(* CODESYS project bentonite_feeder

Project tree, tasks and I/O mapping:
  ecomatDisplay43inch_64bit_1 : ecomatDisplay43inch_64bit, ifm electronic, order no. 
      , version 3.5.19.4
    application Application
      libraries: CmpBitmapPool, * (System); ifmDevice_ecomatDisplay, * (ifm electronic); Datasource Symbolic Access, * (3S - Smart Software Solutions GmbH); Standard, 3.5.18.0 (System); Util, 3.5.19.0 (System)
      task control_task (cyclic, interval 2 ms, priority 17) calls control_prg
      task VISU_TASK (cyclic, interval 5 ms, priority 31) calls VisuElems.Visu_Prg, ifm_device
      control/
        function calc_smoothing [ST]
        program control_prg [CFC]
        function block fb_SlurryPump [LD]: calculate_time
        function block fb_TOI [ST]
        function block PV7603 [ST]
      hmi/
        d pad/
          function block d_pad_fb [ST]: down, left, right, switch_visu, up
        program ifm_device [ST]
        image pool ImagePool
        interfaces/
          function block selectable_item_base [ST]: hover, item_action, leave, select
        menu objects/
          dummy item/
            visualisation dummy_item
            function block fb_dummy_item [ST]: fb_Init, item_action
          hamburger/
            function block fb_hamburger_item [ST]: close, fb_Init, item_action
            visualisation hamburger
          menu data/
            visualisation Empty_visu_reference
            global variables g_menu_colors
            image pool menu_pool
            data type nav_item_enum
          menu item/
            function block fb_menu_item [ST]: fb_Init, item_action
            visualisation menu_item
          toggle items/
            integer setting/
              function block fb_integer_setting [ST]: decrease, fb_Init, increase, item_action, leave
              visualisation integer_setting_dialog
              visualisation integer_setting_item
            number selector/
            real setting/
              function block fb_real_setting [ST]: decrease, fb_Init, increase, item_action, leave
              visualisation real_setting_item
            visualisation toggle_item
        visualisation Parameters
        visualisation Test_Frame_2
        visualisation Test_Frame_3
        visualisation Test_Frame_4
        visualisation Test_Frame_5
        visualisation Test_Frame
      global variables pr
      visualisation Test_Visu
    Communication : Communication, ifm electronic, version 3.5.19.4
      CAN : CAN, ifm electronic, version 3.5.19.4
      Ethernet : Ethernet, ifm electronic, version 3.5.19.4
  5ce3da45-db07-42e7-a21c-a00fff4ed8f6|C:\Users\johnm\Downloads\Full-Circle-Logo-HorizStack.png
  5ce3da45-db07-42e7-a21c-a00fff4ed8f6|C:\Users\johnm\Downloads\Full-Circle-Logo-HorizStack.png
  5ce3da45-db07-42e7-a21c-a00fff4ed8f6|C:\Users\johnm\Full Circle Water\Controls - Documents\Software Versions\graphics\Full Circle Logos (new)\Horizontal\Full-Circle-Logo-Horizontal.png
  5ce3da45-db07-42e7-a21c-a00fff4ed8f6|C:\Users\johnm\Pictures\analytics icon.png
  5ce3da45-db07-42e7-a21c-a00fff4ed8f6|C:\Users\johnm\Pictures\analytics icon.png
  5ce3da45-db07-42e7-a21c-a00fff4ed8f6|C:\Users\johnm\Pictures\analytics icon.png
  5ce3da45-db07-42e7-a21c-a00fff4ed8f6|C:\Users\johnm\Pictures\analytics icon.png
  5ce3da45-db07-42e7-a21c-a00fff4ed8f6|C:\Users\johnm\Pictures\analytics icon.png
  5ce3da45-db07-42e7-a21c-a00fff4ed8f6|C:\Users\johnm\Pictures\analytics icon.png
  5ce3da45-db07-42e7-a21c-a00fff4ed8f6|C:\Users\johnm\Pictures\analytics icon.png
  text list GlobalTextList
  visualisation Visualization
*)

// ecomatDisplay43inch_64bit_1/Application/hmi/menu objects/menu data/nav_item_enum
{attribute 'qualified_only'}
{attribute 'strict'}
TYPE nav_item_enum :
(
	hover:= 0,
	select:= 1,
	selected:= 2,
	leave:= 3, 
	accent:= 4,
	alarm:= 5
);
END_TYPE

// ecomatDisplay43inch_64bit_1/Application/pr
{attribute 'qualified_only'}
VAR_GLOBAL PERSISTENT RETAIN
	//parameter list
	pump_gpm: UINT;
	dose_trigger: UINT; //gallons
	dose_amount: REAL; //pounds with 1 decimal
	charge_time: UINT; //time
	sensor_setpoint: UINT;
	psi_threshold: UINT;
	psi_debounce: UINT; //time
	flow_back: UINT; //amount of gal backfeeding on pump-off
END_VAR

// ecomatDisplay43inch_64bit_1/Application/hmi/menu objects/menu data/g_menu_colors
{attribute 'qualified_only'}
VAR_GLOBAL
	default: DWORD:= 16#FF2C323F;
	nav: ARRAY [nav_item_enum.hover..nav_item_enum.alarm] OF DWORD:= 
		[16#FF464C57, 16#FF7B7F87, 16#FF7B7F87, 16#FF2C323F, 16#FF89A1D3];
	//each position contains corresponding color
	//declare local variable of type 'nav_item_enum,' (ex. 'nav_command') and pass g_menu_colors.nav[nav_command] to the element
END_VAR

// ecomatDisplay43inch_64bit_1/Application/control/control_prg
PROGRAM control_prg
VAR
	simu_toi: fb_TOI; 
	simu_in: BOOL; 
	simu_reset: BOOL;
	tmr: TON; 
END_VAR

simu_toi(IN := simu_in, RESET := simu_reset, PT := T#20s); // FB_TOI

END_PROGRAM

// ecomatDisplay43inch_64bit_1/Application/control/fb_TOI
FUNCTION_BLOCK fb_TOI

VAR_INPUT
	IN: BOOL;
	RESET: BOOL;
	PT: TIME;
END_VAR

VAR_OUTPUT
	ET: TIME;
	Q: BOOL;
END_VAR

VAR
	Start_Time: TIME;
	Saved_Time: TIME;
	RT_IN: R_TRIG;
END_VAR

RT_IN(
	CLK:= IN,
	Q=>,
);

IF RESET THEN 
	ET:= T#0MS;
	Saved_Time:= T#0MS; //reset the time output
END_IF

IF RT_IN.Q THEN
	Start_Time:= TIME(); //when in triggers keep track of time
	Saved_Time:= ET; //and "save" the output time
END_IF

IF IN THEN
	ET:= Saved_Time + TIME() - Start_Time; 
END_IF //output time is saved time and counts from when IN triggered

Q:= ET >= PT; //q is true when output time is above PT

END_FUNCTION_BLOCK

// ecomatDisplay43inch_64bit_1/Application/hmi/ifm_device
PROGRAM ifm_device

VAR
	Reset_Keys: ifmDevice.ResetKeyMapping;
	Key_Map: ifmDevice.SetKeyMapping;
	KeyMapping: ifmDevice.stKEY_MAP_LIST;
	test: BOOL;
END_VAR

VAR
	Start_up_done: BOOL:= 0;
END_VAR

KeyMapping.eKey2_Up:=  		ifmDevice.eKEY_MAP_CODES.LEFT;
KeyMapping.eKey2_Down:=		ifmDevice.eKEY_MAP_CODES.RIGHT;
KeyMapping.eKey2_Left:=		ifmDevice.eKEY_MAP_CODES.DOWN;
KeyMapping.eKey2_Right:=	ifmDevice.eKEY_MAP_CODES.UP;
KeyMapping.eKey2_Return:=	ifmDevice.eKEY_MAP_CODES.SPACE;
		
Reset_Keys(
	xExecute:= NOT(Start_up_done AND test),
	xDone=>,
	xError=>,
	eDiagInfo=>
);

Key_Map(
	xExecute:= NOT(start_up_done AND test),
	xDone=>,
	xError=>,
	eDiagInfo=>,
	stKeyMapList:= KeyMapping,
);

test:= Start_up_done;
Start_up_done S= Reset_Keys.xDone AND Key_Map.xDone;

END_PROGRAM

// ecomatDisplay43inch_64bit_1/Application/control/calc_smoothing
FUNCTION calc_smoothing : REAL
VAR_INPUT
	cycle_time: TIME;
	time_constant: TIME:= T#2MS; 
END_VAR
VAR CONSTANT
	
END_VAR

calc_smoothing:= 1 - EXPT(2.71828, (-1.0 * (TO_REAL(cycle_time)) / TO_REAL(time_constant)));

END_FUNCTION

// ecomatDisplay43inch_64bit_1/Application/control/fb_SlurryPump
FUNCTION_BLOCK fb_SlurryPump

VAR_INPUT
	pumping: BOOL;
	gpm: UINT;
	trigger_volume: UINT;
END_VAR

VAR_OUTPUT
	dose: BOOL; //single shot
END_VAR

VAR
	flow_counter: REAL;
	time_val: TIME;
	timer_fb: fb_TOI;
END_VAR

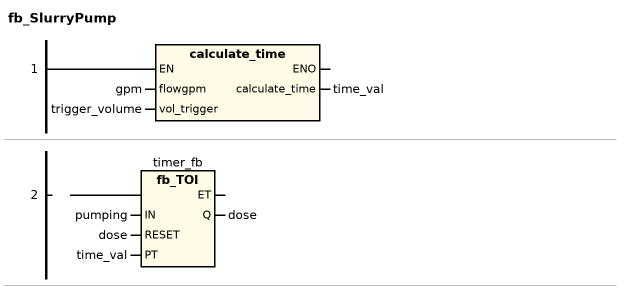
// NETWORK 1
time_val := calculate_time(flowgpm := gpm, vol_trigger := trigger_volume);

// NETWORK 2
timer_fb(IN := pumping, RESET := dose, PT := time_val, Q => dose); // fb_TOI

METHOD calculate_time : TIME
VAR_INPUT
	flowgpm: UINT;
	vol_trigger: UINT;
END_VAR

VAR CONSTANT
	min_to_ms: UINT:= 60000;
END_VAR
calculate_time:= TO_TIME(
	TO_UINT(
		TO_REAL(vol_trigger) 
	/ 	TO_REAL(flowgpm) //calc how many minutes
	* 	min_to_ms) //convert to ms
);
END_METHOD

END_FUNCTION_BLOCK

// ecomatDisplay43inch_64bit_1/Application/control/PV7603
FUNCTION_BLOCK PV7603
VAR_INPUT
	IOL_Read: ARRAY [0..3] OF WORD;
	time_setting: TIME;
END_VAR
VAR_OUTPUT
END_VAR
VAR
	factor: REAL;
	cycle_time: TIME;
	filtered_val: REAL;
	raw_signal: REAL;
END_VAR

raw_signal:= TO_REAL(IOL_Read[0]);

factor := calc_smoothing(T#2MS, time_setting);

filtered_val:= 
	(filtered_val * (1.0 - factor)) 
+ 	(raw_signal * factor);

END_FUNCTION_BLOCK

// ecomatDisplay43inch_64bit_1/Application/hmi/d pad/d_pad_fb
FUNCTION_BLOCK d_pad_fb
VAR_INPUT CONSTANT
	x_bounds: UINT:= 3;
END_VAR
VAR_INPUT
	disable_nav: BOOL;
	y_bounds: ARRAY [0..20] OF UINT;
END_VAR

VAR_OUTPUT
	position: ARRAY [0..1] OF UINT:= [1, 0];
END_VAR

METHOD down
VAR_INPUT
END_VAR
IF THIS^.disable_nav THEN
	RETURN; 
END_IF

IF THIS^.y_bounds[position[0]] > THIS^.position[1] THEN
	THIS^.position[1]:= THIS^.position[1] + 1;
END_IF
END_METHOD

METHOD left
VAR_INPUT
END_VAR
IF THIS^.disable_nav THEN
	RETURN; 
END_IF

IF THIS^.x_bounds > THIS^.position[0] THEN
	THIS^.position[0]:= THIS^.position[0] + 1;
	THIS^.position[1]:= 0;
END_IF
END_METHOD

METHOD right
VAR_INPUT
END_VAR
IF THIS^.disable_nav THEN
	RETURN; 
END_IF

IF THIS^.position[0] < 1 THEN
	RETURN;
END_IF

THIS^.position[0]:= THIS^.position[0] - 1;
THIS^.position[1]:= 0;
END_METHOD

METHOD switch_visu
VAR_INPUT
END_VAR
THIS^.position[0]:= 0;
THIS^.position[1]:= 0;
END_METHOD

METHOD up
VAR_INPUT
END_VAR
IF THIS^.disable_nav THEN
	RETURN; 
END_IF

IF THIS^.position[1] < 1 THEN
	RETURN;
END_IF

THIS^.position[1]:= THIS^.position[1] - 1;
END_METHOD

END_FUNCTION_BLOCK

// ecomatDisplay43inch_64bit_1/Application/hmi/interfaces/selectable_item_base
FUNCTION_BLOCK ABSTRACT selectable_item_base
VAR_INPUT
	position: ARRAY [0..1] OF UINT;
END_VAR
VAR_OUTPUT
END_VAR
VAR
	color: DWORD:= 16#FFFFFFFF;
END_VAR

METHOD hover
THIS^.color:= g_menu_colors.nav[nav_item_enum.hover];
//changes fb 'color' to menu color value for hover action
END_METHOD

METHOD ABSTRACT item_action
END_METHOD

METHOD leave
VAR_INPUT
END_VAR
THIS^.color:= g_menu_colors.nav[nav_item_enum.leave];
//changes fb 'color' to menu color value for hover action
END_METHOD

METHOD select
THIS^.color:= g_menu_colors.nav[nav_item_enum.select];
//changes fb 'color' to menu color value for selected action
THIS^.item_action();
END_METHOD

END_FUNCTION_BLOCK

// ecomatDisplay43inch_64bit_1/Application/hmi/menu objects/dummy item/fb_dummy_item
FUNCTION_BLOCK fb_dummy_item EXTENDS selectable_item_base
VAR_INPUT
END_VAR
VAR_OUTPUT
END_VAR
VAR
END_VAR

//FB_Init is always available implicitly and it is used primarily for initialization.
//The return value is not evaluated. For a specific influence, you can also declare the
//methods explicitly and provide additional code there with the standard initialization
//code. You can evaluate the return value.
METHOD FB_Init: BOOL
VAR_INPUT
    bInitRetains: BOOL; // TRUE: the retain variables are initialized (reset warm / reset cold)
    bInCopyCode: BOOL:= TRUE;  // TRUE: the instance will be copied to the copy code afterward (online change)   
END_VAR
THIS^.color:= g_menu_colors.default;
END_METHOD

METHOD item_action
END_METHOD

END_FUNCTION_BLOCK

// ecomatDisplay43inch_64bit_1/Application/hmi/menu objects/hamburger/fb_hamburger_item
FUNCTION_BLOCK fb_hamburger_item EXTENDS selectable_item_base
VAR_INPUT
END_VAR
VAR_OUTPUT
	open: BOOL;
END_VAR

METHOD close : BOOL
VAR_INPUT
END_VAR
THIS^.open:= 0;
END_METHOD

//FB_Init is always available implicitly and it is used primarily for initialization.
//The return value is not evaluated. For a specific influence, you can also declare the
//methods explicitly and provide additional code there with the standard initialization
//code. You can evaluate the return value.
METHOD FB_Init: BOOL
VAR_INPUT
    bInitRetains: BOOL; // TRUE: the retain variables are initialized (reset warm / reset cold)
    bInCopyCode: BOOL:= TRUE;  // TRUE: the instance will be copied to the copy code afterward (online change)   
END_VAR
THIS^.color:= g_menu_colors.default;
END_METHOD

METHOD item_action
THIS^.open:= 1;
END_METHOD

END_FUNCTION_BLOCK

// ecomatDisplay43inch_64bit_1/Application/hmi/menu objects/menu item/fb_menu_item
FUNCTION_BLOCK fb_menu_item	EXTENDS selectable_item_base
(*Visualizations of 'menu items,' code implementation using references contained here.*)
(*All implementation is done using the fb methods, and are called in visualization.*)
VAR_INPUT
	visu_reference: REFERENCE TO UINT;
	(*index of configured frame visu*)
	(*and order in list - d pad navigation*)
END_VAR
VAR_OUTPUT
END_VAR

//FB_Init is always available implicitly and it is used primarily for initialization.
//The return value is not evaluated. For a specific influence, you can also declare the
//methods explicitly and provide additional code there with the standard initialization
//code. You can evaluate the return value.
METHOD FB_Init: BOOL
VAR_INPUT
    bInitRetains: BOOL; // TRUE: the retain variables are initialized (reset warm / reset cold)
    bInCopyCode: BOOL:= TRUE;  // TRUE: the instance will be copied to the copy code afterward (online change)   
END_VAR
THIS^.color:= g_menu_colors.default;
END_METHOD

METHOD item_action
THIS^.visu_reference:= THIS^.position[1] - 1;
(*assign index to the frame*)
END_METHOD

END_FUNCTION_BLOCK

// ecomatDisplay43inch_64bit_1/Application/hmi/menu objects/toggle items/integer setting/fb_integer_setting
FUNCTION_BLOCK fb_integer_setting EXTENDS selectable_item_base
VAR_INPUT
	integer: REFERENCE TO UINT;
	increment: UINT;
	default: UINT;
	max_value: UINT;
	min_value: UINT;
END_VAR
VAR_OUTPUT
	selected: BOOL;

END_VAR
VAR
	int_array: ARRAY [0..4] OF UINT; // ones, tens, hundreds, thousands, ten-thousands
END_VAR

METHOD decrease
VAR_INPUT
END_VAR
IF THIS^.integer - THIS^.increment >= THIS^.min_value THEN
	THIS^.integer:= THIS^.integer - THIS^.increment;
END_IF
END_METHOD

(*FB_Init is always available implicitly and it is used primarily for initialization.
The return value is not evaluated. For a specific influence, you can also declare the
methods explicitly and provide additional code there with the standard initialization
code. You can evaluate the return value.*)
METHOD FB_Init : BOOL
VAR_INPUT
	(* TRUE: the retain variables are initialized (reset warm / reset cold)*)
	bInitRetains	: BOOL;
	(* TRUE: the instance will be copied to the copy code afterward (online change)   *)
	bInCopyCode	: BOOL := TRUE;
END_VAR
THIS^.color:= g_menu_colors.default;
(*
THIS^.int_array[0]:= THIS^.integer / 1		MOD 10;
THIS^.int_array[1]:= THIS^.integer / 10		MOD 10;
THIS^.int_array[2]:= THIS^.integer / 100	MOD 10;
THIS^.int_array[3]:= THIS^.integer / 1000	MOD 10;
THIS^.int_array[4]:= THIS^.integer / 10000	MOD 10;*)
END_METHOD

METHOD increase
VAR_INPUT
END_VAR
IF THIS^.integer + THIS^.increment <= THIS^.max_value THEN
	THIS^.integer:= THIS^.integer + THIS^.increment;
END_IF
END_METHOD

METHOD item_action
VAR_INPUT
END_VAR
THIS^.selected:= THIS^.selected XOR TRUE;
IF NOT THIS^.selected THEN
	THIS^.hover();
END_IF
END_METHOD

METHOD leave
VAR_INPUT
END_VAR
THIS^.color:= g_menu_colors.nav[nav_item_enum.leave];
//changes fb 'color' to menu color value for hover action
THIS^.selected:= 0;
END_METHOD

END_FUNCTION_BLOCK

// ecomatDisplay43inch_64bit_1/Application/hmi/menu objects/toggle items/real setting/fb_real_setting
FUNCTION_BLOCK fb_real_setting EXTENDS selectable_item_base
VAR_INPUT
	real_var: REFERENCE TO REAL;
	increment: REAL;
	max_value: REAL;
	min_value: REAL;
END_VAR
VAR_OUTPUT
	selected: BOOL;
END_VAR
VAR
END_VAR

METHOD decrease
VAR_INPUT
END_VAR
IF THIS^.real_var - THIS^.increment >= THIS^.min_value THEN
	THIS^.real_var:= THIS^.real_var - THIS^.increment;
END_IF
END_METHOD

//FB_Init is always available implicitly and it is used primarily for initialization.
//The return value is not evaluated. For a specific influence, you can also declare the
//methods explicitly and provide additional code there with the standard initialization
//code. You can evaluate the return value.
METHOD FB_Init: BOOL
VAR_INPUT
    bInitRetains: BOOL; // TRUE: the retain variables are initialized (reset warm / reset cold)
    bInCopyCode: BOOL:= TRUE;  // TRUE: the instance will be copied to the copy code afterward (online change)   
END_VAR
THIS^.color:= g_menu_colors.default;
END_METHOD

METHOD increase
VAR_INPUT
END_VAR
IF THIS^.real_var + THIS^.increment <= THIS^.max_value THEN
	THIS^.real_var:= THIS^.real_var + THIS^.increment;
END_IF
END_METHOD

METHOD item_action
VAR_INPUT
END_VAR
THIS^.selected:= THIS^.selected XOR TRUE;
IF NOT THIS^.selected THEN
	THIS^.hover();
END_IF
END_METHOD

METHOD leave
VAR_INPUT
END_VAR
THIS^.color:= g_menu_colors.nav[nav_item_enum.leave];
//changes fb 'color' to menu color value for hover action
THIS^.selected:= 0;
END_METHOD

END_FUNCTION_BLOCK

// /Visualization
VISUALIZATION Visualization  // 1024x768
END_VISUALIZATION

// ecomatDisplay43inch_64bit_1/Application/Test_Visu
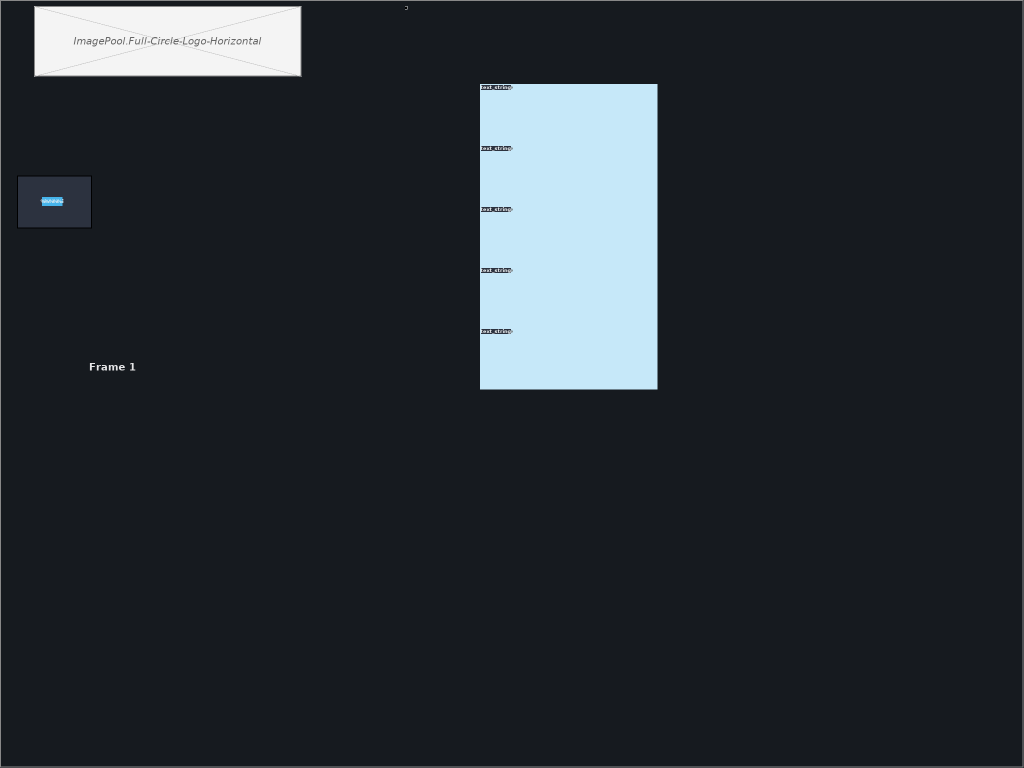
VISUALIZATION Test_Visu  // 1024x768
VAR
	screen_index: UINT:= 0;
	selected_index: UINT;
	
	d_pad: d_pad_fb:= (x_bounds:= 2, y_bounds:= [5, 7]);
	
	hamburger_item: fb_hamburger_item:= (position:= [0,0]);
	test_item:  fb_menu_item:= (visu_reference:= screen_index, position:= [0,1]);
	test_item2: fb_menu_item:= (visu_reference:= screen_index, position:= [0,2]);
	test_item3: fb_menu_item:= (visu_reference:= screen_index, position:= [0,3]);
	test_item4: fb_menu_item:= (visu_reference:= screen_index, position:= [0,4]);
	test_item5: fb_menu_item:= (visu_reference:= screen_index, position:= [0,5]);
	test_item6: fb_menu_item:= (visu_reference:= screen_index, position:= [0,6]);
	
	
	//speed 1 or 2 
	//speed 1 pounds per minute
	//speed 2 pounds per minute
	//enable buzzer for ... 
	
END_VAR
    Frame (0,90 480x710), frame switch variable: screen_index
        shows Test_Frame(d_pad_ref := d_pad)
        shows Parameters(d_pad_ref := d_pad)
        shows Test_Frame_2()
        shows Test_Frame_3()
        shows Test_Frame_4()
        shows Test_Frame_5()
    Rectangle (480,84 177x305)
        p3560616238: -179 * TO_INT(hamburger_item.open)
    Frame (481,85 175x60)
        shows menu_item(Text := Operation, Position := 0, fb_ref := test_item, d_pad_pos := d_pad.position)
        p3560616238: -178 * TO_INT(hamburger_item.open)
    Frame (481,146 175x60)
        shows menu_item(Text := Parameters, Position := 0, fb_ref := test_item2, d_pad_pos := d_pad.position)
        p3560616238: -178 * TO_INT(hamburger_item.open)
    Frame (481,207 175x60)
        shows menu_item(Text := Calibration, Position := 0, fb_ref := test_item3, d_pad_pos := d_pad.position)
        p3560616238: -178 * TO_INT(hamburger_item.open)
    Frame (481,268 175x60)
        shows menu_item(Text := Manual, Position := 0, fb_ref := test_item4, d_pad_pos := d_pad.position)
        p3560616238: -178 * TO_INT(hamburger_item.open)
    Frame (481,329 175x60)
        shows menu_item(Text := Event log, Position := 0, fb_ref := test_item5, d_pad_pos := d_pad.position)
        p3560616238: -178 * TO_INT(hamburger_item.open)
    Frame (405,6 70x70)
        shows hamburger(fb_ref := hamburger_item, d_pad_pos := d_pad.position)
    Image (34,6 267x70), image: ImagePool.Full-Circle-Logo-Horizontal
    hotkey  Id=481042628608, Key=KeyDown=True, KeyName=right, ActionToExecute=Action=STSnippet=d_pad.right();, VisuElemId=-1
    hotkey  Id=481041580032, Key=KeyDown=True, KeyName=left, ActionToExecute=Action=STSnippet=d_pad.left(); IF d_pad.position[0] <> 0 THEN hamburger_item.close(); END_IF, VisuElemId=-1
    hotkey  Id=481040531456, Key=KeyDown=True, KeyName=up, ActionToExecute=Action=STSnippet=d_pad.up();, VisuElemId=-1
    hotkey  Id=481039482880, Key=KeyDown=True, KeyName=down, ActionToExecute=Action=STSnippet=d_pad.down();, VisuElemId=-1
    hotkey  Id=481044725760, Key=KeyDown=True, KeyName=space, VisuElemId=-1
    hotkey  Id=481045774336, Key=KeyDown=True, KeyName=F2, ActionToExecute=Action=STSnippet=hamburger_item.select();, VisuElemId=-1
END_VISUALIZATION

// ecomatDisplay43inch_64bit_1/Application/hmi/Parameters
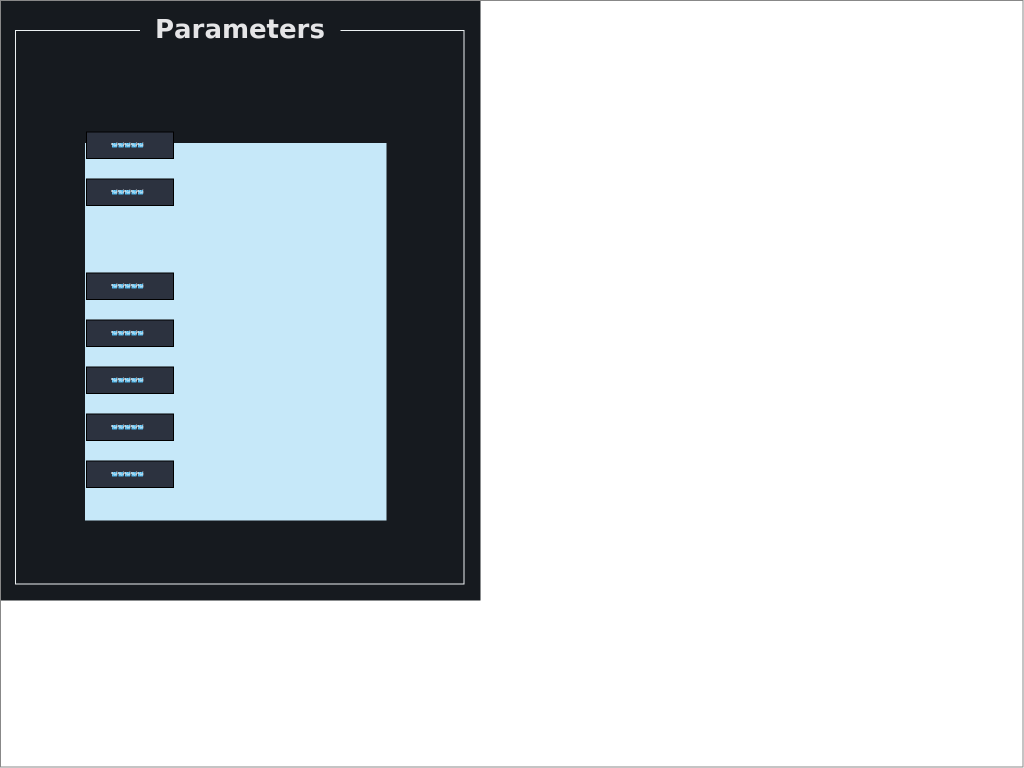
VISUALIZATION Parameters  // 1024x768
VAR_INPUT
	d_pad_ref: REFERENCE TO d_pad_fb; 
END_VAR
VAR
	item_pump_flow: 		fb_integer_setting:=	(position:= [1,0], integer:= pr.pump_gpm, 		increment:= 1, 	max_value:= 100, 	min_value:= 0);
	item_dose_trig: 		fb_integer_setting:=	(position:= [1,1], integer:= pr.dose_trigger, 	increment:= 5, 	max_value:= 10000, 	min_value:= 0);
	item_dose_amount:		fb_real_setting:=		(position:= [1,2], real_var:= pr.dose_amount, 	increment:= 0.1,max_value:= 10, 	min_value:= 0);
	item_charge_time:		fb_integer_setting:=	(position:= [1,3], integer:= pr.charge_time, 	increment:= 1, 	max_value:= 1000, 	min_value:= 0);
	item_sensor_setpoint: 	fb_integer_setting:= 	(position:= [1,4], integer:= pr.sensor_setpoint,increment:= 50, max_value:= 1450,	min_value:= 0);
	item_psi_threshold:		fb_integer_setting:=	(position:= [1,5], integer:= pr.psi_threshold, 	increment:= 1, 	max_value:= 150, 	min_value:= 0); 
	item_psi_debounce:		fb_integer_setting:=	(position:= [1,6], integer:= pr.psi_debounce, 	increment:= 50, max_value:= 2000, 	min_value:= 0);
	item_flow_back:			fb_integer_setting:=	(position:= [1,7], integer:= pr.flow_back,		increment:= 1,	max_value:= 500, 	min_Value:= 0);	
END_VAR
    Rectangle (0,0 480x600)
    RoundedRectangle (15,30 449x554)
    Rectangle (85,143 301x377), invisible if: d_pad_ref.disable_nav
    Frame (86,145 300x144)
        shows integer_setting_item(Name := 'Pump flow', Units := 'gpm', fb_ref := item_pump_flow, ref_d_pad := d_pad_ref)
    Frame (86,333 300x144)
        shows integer_setting_item(Name := 'Material sensor', Units := '', fb_ref := item_sensor_setpoint, ref_d_pad := d_pad_ref)
    Frame (86,192 300x144)
        shows integer_setting_item(Name := 'Dose trigger', Units := 'gal.', fb_ref := item_dose_trig, ref_d_pad := d_pad_ref)
    Frame (86,380 300x144)
        shows integer_setting_item(Name := 'Pumping trigger', Units := 'psi', fb_ref := item_psi_threshold, ref_d_pad := d_pad_ref)
    Frame (86,427 300x144)
        shows integer_setting_item(Name := 'PSI debounce', Units := 'ms', fb_ref := item_psi_debounce, ref_d_pad := d_pad_ref)
    Frame (86,286 300x144)
        shows integer_setting_item(Name := 'Charging time', Units := 'sec', fb_ref := item_charge_time, ref_d_pad := d_pad_ref)
    Frame (86,474 300x144)
        shows integer_setting_item(Name := 'Flow back volume', Units := 'gal.', fb_ref := item_flow_back, ref_d_pad := d_pad_ref)
    Rectangle (140,5 200x48), "Parameters"
END_VISUALIZATION

// ecomatDisplay43inch_64bit_1/Application/hmi/Test_Frame_2
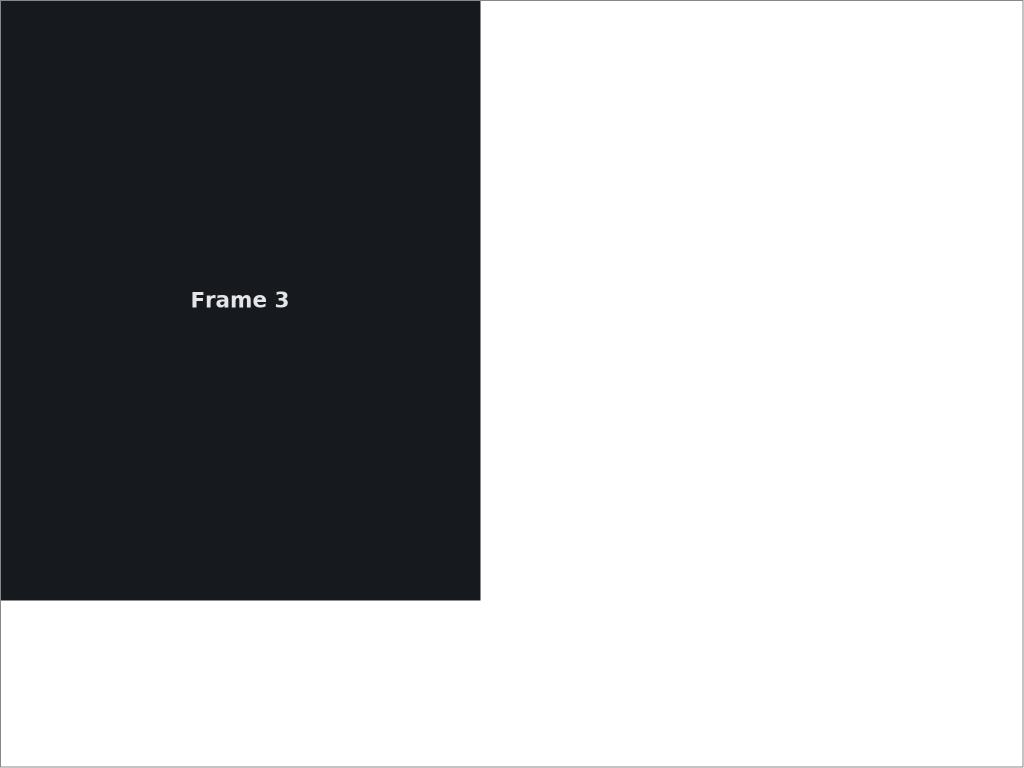
VISUALIZATION Test_Frame_2  // 1024x768
VAR_INPUT
	SELECTED: BOOL;
END_VAR
    Rectangle (0,0 480x600), "Frame 3", colour variable: g_menu_colors.default
        p3450524324: g_menu_colors.default
END_VISUALIZATION

// ecomatDisplay43inch_64bit_1/Application/hmi/Test_Frame_3
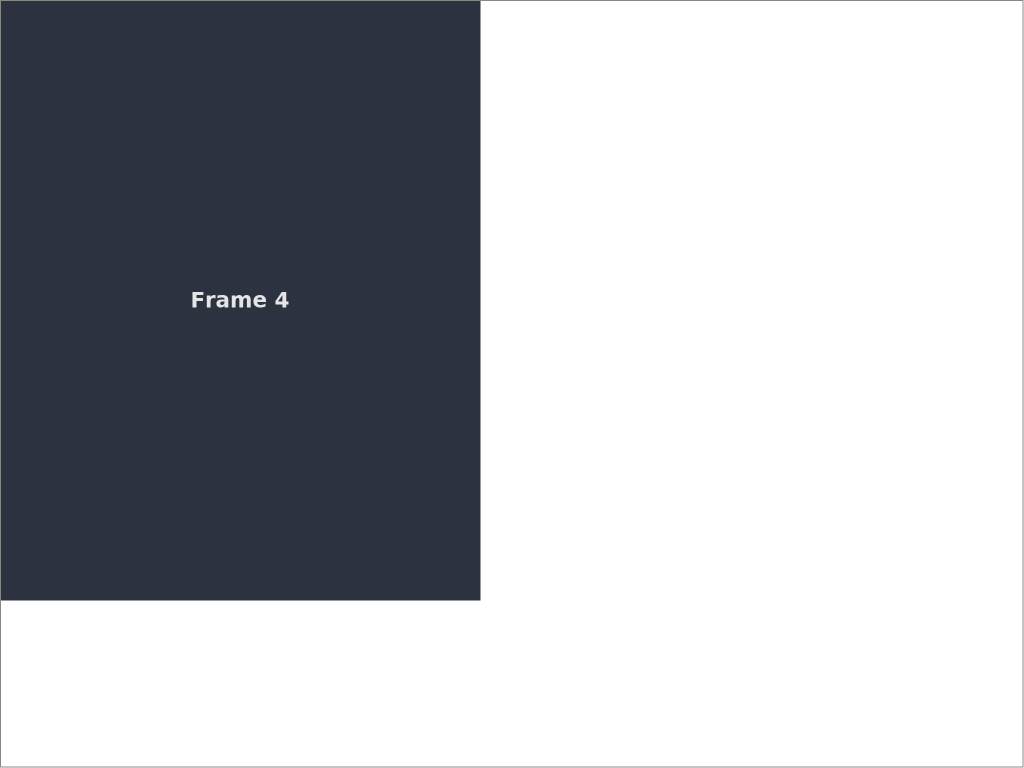
VISUALIZATION Test_Frame_3  // 1024x768
VAR_INPUT
	SELECTED: BOOL;
END_VAR
    Rectangle (0,0 480x600), "Frame 4", colour variable: g_menu_colors.default
        p3450524324: g_menu_colors.default
END_VISUALIZATION

// ecomatDisplay43inch_64bit_1/Application/hmi/Test_Frame_4
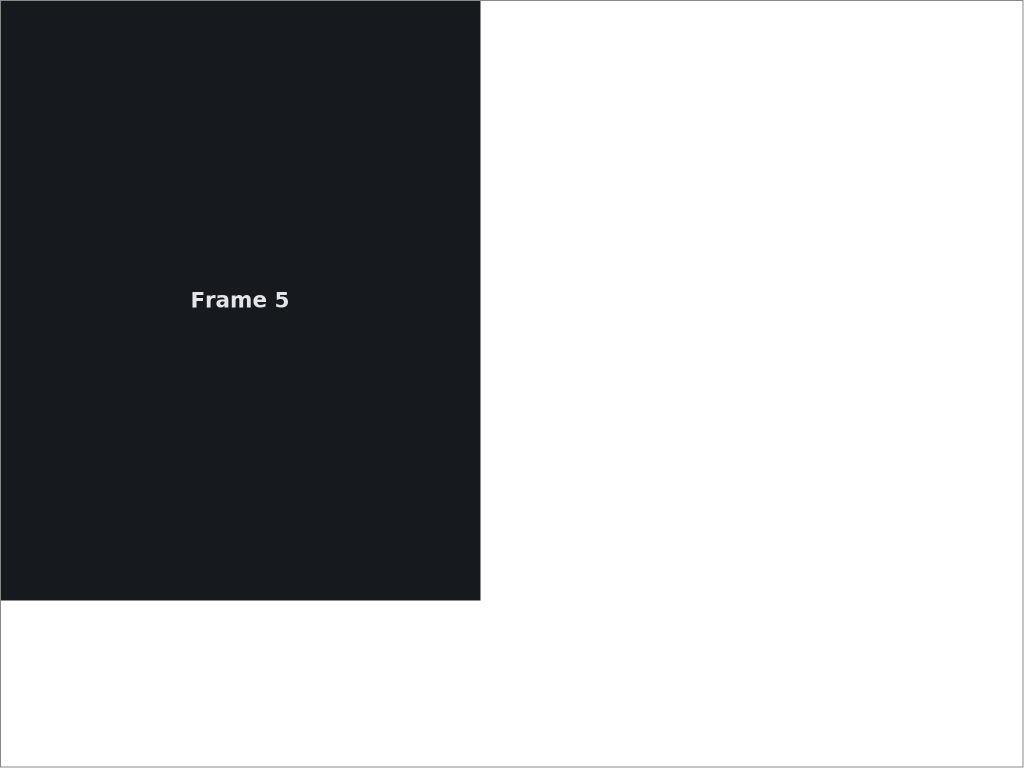
VISUALIZATION Test_Frame_4  // 1024x768
VAR_INPUT
	SELECTED: BOOL;
END_VAR
    Rectangle (0,0 480x600), "Frame 5", colour variable: g_menu_colors.default
        p3450524324: g_menu_colors.default
END_VISUALIZATION

// ecomatDisplay43inch_64bit_1/Application/hmi/Test_Frame_5
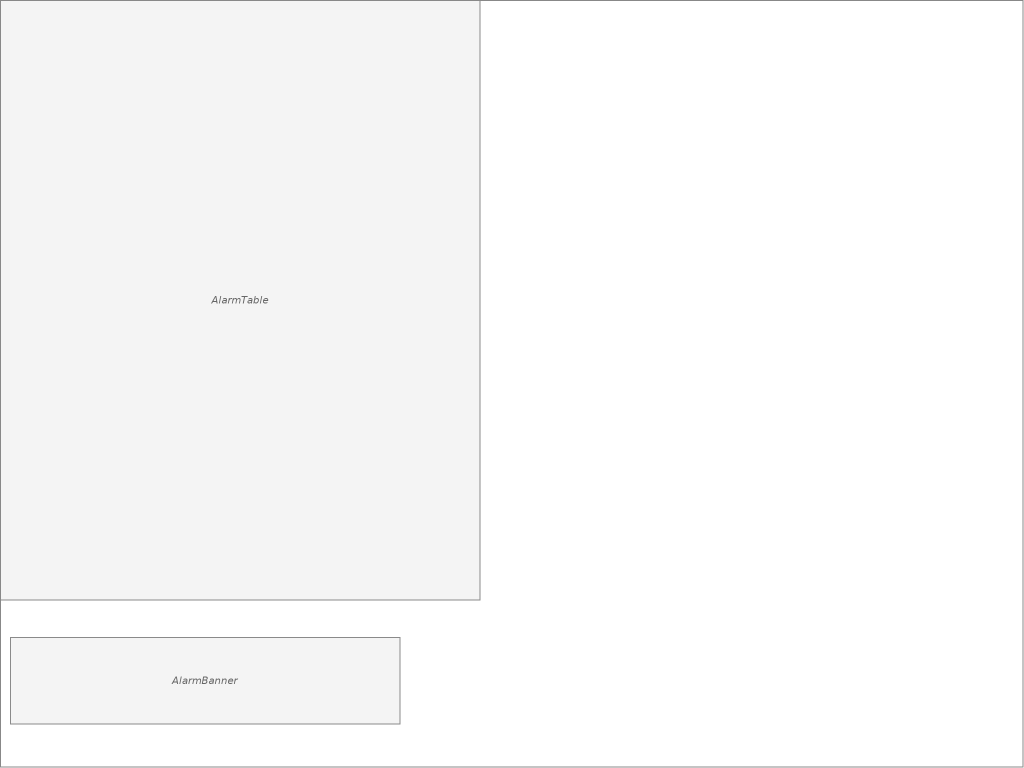
VISUALIZATION Test_Frame_5  // 1024x768
VAR_INPUT
	SELECTED: BOOL;
END_VAR
    Rectangle (0,0 480x600), "Frame 6", colour variable: g_menu_colors.default
        p3450524324: g_menu_colors.default
    AlarmTable (0,0 480x600)
        p1521930926: __All
        p1663851261: __All
    AlarmBanner (10,637 390x87)
        p1521930926: __All
        p1663851261: __All
END_VISUALIZATION

// ecomatDisplay43inch_64bit_1/Application/hmi/Test_Frame
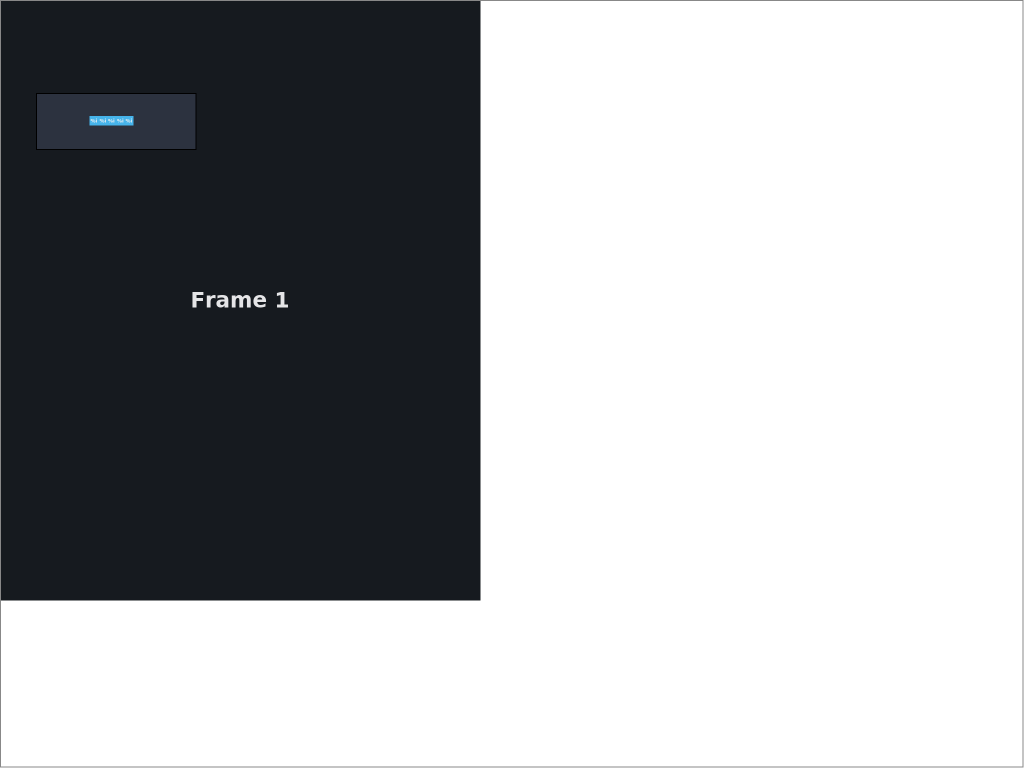
VISUALIZATION Test_Frame  // 1024x768
VAR
		item_dose_trig: fb_integer_setting:=	(
			position:= [1,1], 
			integer:= pr.dose_trigger, 	
			increment:= 5, 
			max_value:= 100, 	
			min_value:= 0
		);
END_VAR
VAR_INPUT
	d_pad_ref: REFERENCE TO d_pad_fb;
END_VAR
    Rectangle (0,0 480x600), "Frame 1"
    Frame (38,96 405x209)
        shows integer_setting_dialog(Name := 'name', Units := 'units', fb_ref := item_dose_trig, ref_d_pad := d_pad_ref)
END_VISUALIZATION

// ecomatDisplay43inch_64bit_1/Application/hmi/menu objects/dummy item/dummy_item
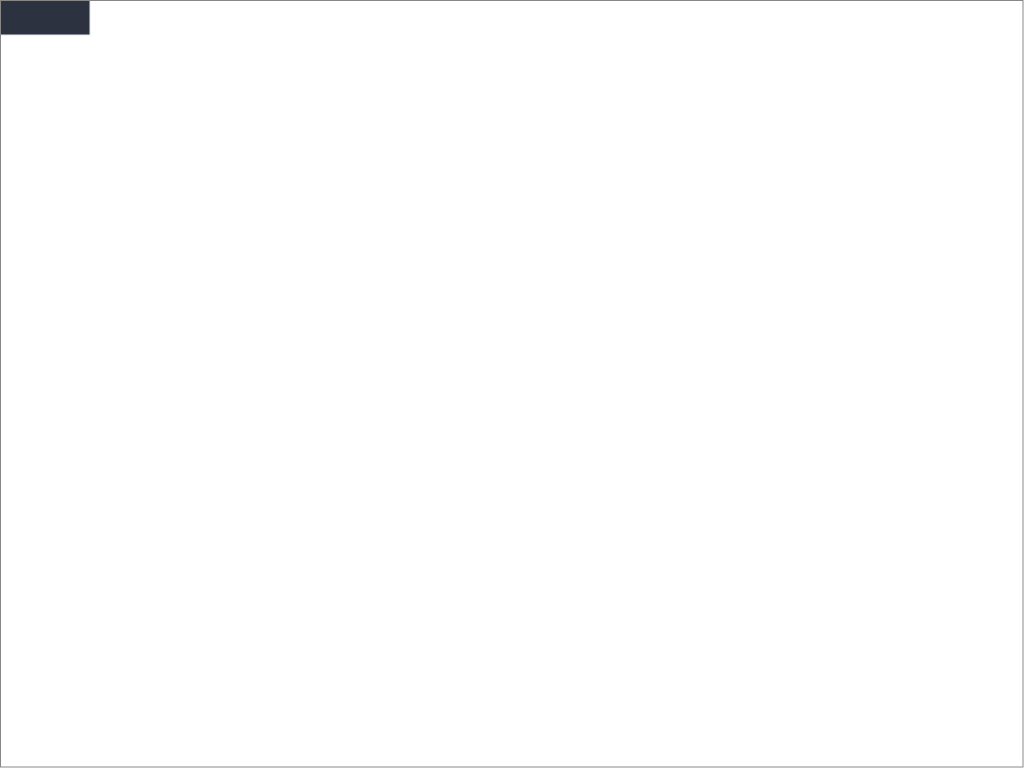
VISUALIZATION dummy_item  // 1024x768
VAR_INPUT
	fb_ref: REFERENCE TO fb_dummy_item;
	d_pad_pos: REFERENCE TO ARRAY [0..1] OF UINT;
END_VAR
    Rectangle (0,0 90x35)
    Rectangle (0,0 90x35)
    Rectangle (0,0 90x35), colour variable: fb_ref.color
        p3450524324: fb_ref.color
        p3092690914: fb_ref.color
        p2167032090: fb_ref.color
        OnMouseClick: execute { fb_ref.select(); }
        OnMouseDown: execute {  }
        OnMouseEnter: execute { fb_ref.hover(); }
        OnMouseLeave: execute { fb_ref.leave(); }
    Rectangle (0,0 90x35), colour toggle: fb_ref.color = g_menu_colors.nav[nav_item_enum.selected], colour variable: fb_ref.color
        p3450524324: g_menu_colors.nav[nav_item_enum.selected]
        p3092690914: g_menu_colors.nav[nav_item_enum.accent]
        p2167032090: fb_ref.color
        OnMouseClick: execute {  }
        OnMouseDown: execute { fb_ref.select(); d_pad_pos:= fb_ref.position; }
        OnMouseEnter: execute { fb_ref.hover(); }
        OnMouseLeave: execute { fb_ref.leave(); }
        OnMouseUp: execute { fb_ref.hover(); }
    hotkey  Id=481040531456, Key=KeyName=right, ActionToExecute=Action=STSnippet=IF d_pad_pos[0] = fb_ref.position[0] AND d_pad_pos[1] = fb_ref.position[1] THEN fb_ref.hover(); END_IF IF NOT(d_pad_pos[0] = fb_ref.position[0] AND d_pad_pos[1] = fb_ref.position[1]) THEN fb_ref.leave(); END_IF, VisuElemId=-1
    hotkey  Id=481039482880, Key=KeyName=left, ActionToExecute=Action=STSnippet=IF d_pad_pos[0] = fb_ref.position[0] AND d_pad_pos[1] = fb_ref.position[1] THEN fb_ref.hover(); END_IF IF NOT(d_pad_pos[0] = fb_ref.position[0] AND d_pad_pos[1] = fb_ref.position[1]) THEN fb_ref.leave(); END_IF, VisuElemId=-1
    hotkey  Id=481038434304, Key=KeyName=up, ActionToExecute=Action=STSnippet=IF d_pad_pos[0] = fb_ref.position[0] AND d_pad_pos[1] = fb_ref.position[1] THEN fb_ref.hover(); END_IF IF NOT(d_pad_pos[0] = fb_ref.position[0] AND d_pad_pos[1] = fb_ref.position[1]) THEN fb_ref.leave(); END_IF, VisuElemId=-1
    hotkey  Id=481037385728, Key=KeyName=down, ActionToExecute=Action=STSnippet=IF d_pad_pos[0] = fb_ref.position[0] AND d_pad_pos[1] = fb_ref.position[1] THEN fb_ref.hover(); END_IF IF NOT(d_pad_pos[0] = fb_ref.position[0] AND d_pad_pos[1] = fb_ref.position[1]) THEN fb_ref.leave(); END_IF, VisuElemId=-1
END_VISUALIZATION

// ecomatDisplay43inch_64bit_1/Application/hmi/menu objects/hamburger/hamburger
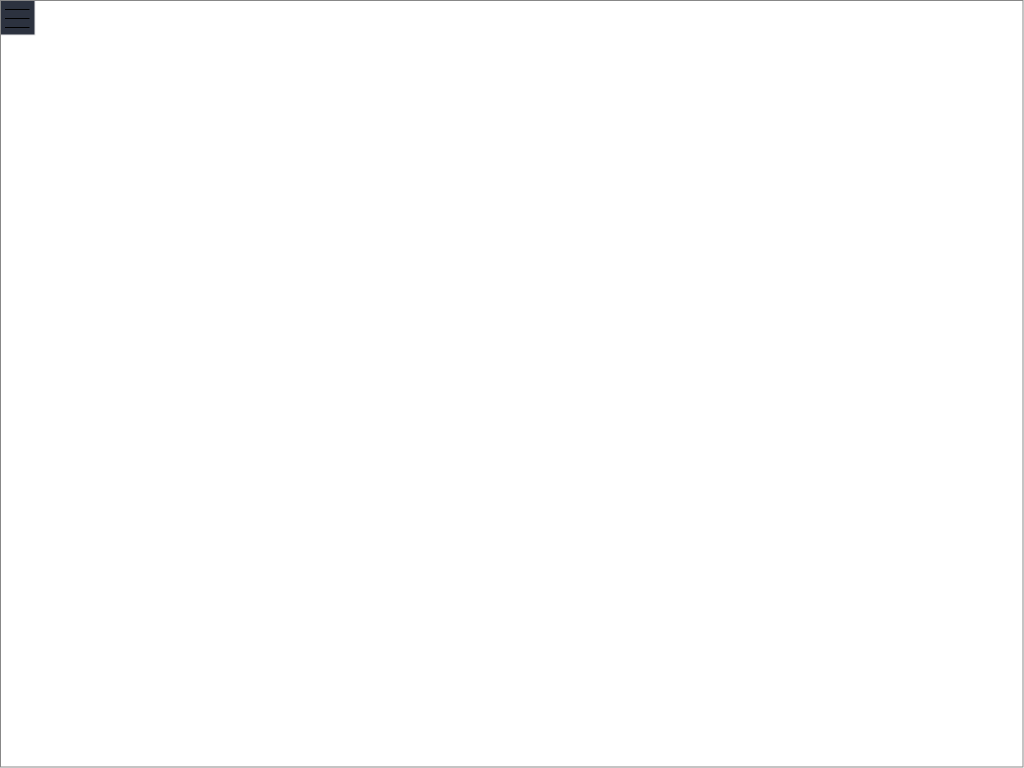
VISUALIZATION hamburger  // 1024x768
VAR_INPUT
	fb_ref: REFERENCE TO fb_hamburger_item;
	d_pad_pos: REFERENCE TO ARRAY [0..1] OF UINT;
END_VAR
    Rectangle (0,0 35x35)
    Rectangle (0,0 35x35)
    Rectangle (0,0 35x35), colour variable: fb_ref.color
        p3450524324: fb_ref.color
        p3092690914: fb_ref.color
        p2167032090: fb_ref.color
        OnMouseClick: execute { fb_ref.select(); }
        OnMouseDown: execute {  }
        OnMouseEnter: execute { fb_ref.hover(); }
        OnMouseLeave: execute { fb_ref.leave(); }
    Rectangle (0,0 35x35), colour toggle: fb_ref.color = g_menu_colors.nav[nav_item_enum.selected], colour variable: fb_ref.color
        p3450524324: g_menu_colors.nav[nav_item_enum.selected]
        p3092690914: g_menu_colors.nav[nav_item_enum.accent]
        p2167032090: g_menu_colors.nav[nav_item_enum.selected]
        OnMouseClick: execute {  }
        OnMouseDown: execute { fb_ref.select(); d_pad_pos:= fb_ref.position; }
        OnMouseEnter: execute { fb_ref.hover(); }
        OnMouseLeave: execute { fb_ref.leave(); }
        OnMouseUp: execute { fb_ref.hover(); }
    Line (5,27) (29,27), colour toggle: fb_ref.color = g_menu_colors.nav[nav_item_enum.selected]
        p2175578022: g_menu_colors.nav[nav_item_enum.selected]
        p573394764: g_menu_colors.nav[nav_item_enum.accent]
    Line (5,18) (29,18), colour toggle: fb_ref.color = g_menu_colors.nav[nav_item_enum.selected]
        p2175578022: g_menu_colors.nav[nav_item_enum.selected]
        p573394764: g_menu_colors.nav[nav_item_enum.accent]
    Line (5,9) (29,9), colour toggle: fb_ref.color = g_menu_colors.nav[nav_item_enum.selected]
        p2175578022: g_menu_colors.nav[nav_item_enum.selected]
        p573394764: g_menu_colors.nav[nav_item_enum.accent]
    hotkey  Id=481040531456, Key=KeyDown=True, KeyName=right, ActionToExecute=Action=STSnippet=IF d_pad_pos[0] = fb_ref.position[0] AND d_pad_pos[1] = fb_ref.position[1] THEN fb_ref.select(); END_IF IF NOT(d_pad_pos[0] = fb_ref.position[0] AND d_pad_pos[1] = fb_ref.position[1]) THEN fb_ref.leave(); fb_ref.close(); END_IF, VisuElemId=-1
    hotkey  Id=481039482880, Key=KeyName=left, ActionToExecute=Action=STSnippet=IF d_pad_pos[0] = fb_ref.position[0] AND d_pad_pos[1] = fb_ref.position[1] THEN fb_ref.select(); END_IF IF NOT(d_pad_pos[0] = fb_ref.position[0] AND d_pad_pos[1] = fb_ref.position[1]) THEN fb_ref.leave(); fb_ref.close(); END_IF, VisuElemId=-1
    hotkey  Id=481038434304, Key=KeyDown=True, KeyName=up, ActionToExecute=Action=STSnippet=IF d_pad_pos[0] = fb_ref.position[0] AND d_pad_pos[1] = fb_ref.position[1] THEN fb_ref.select(); END_IF IF NOT(d_pad_pos[0] = fb_ref.position[0] AND d_pad_pos[1] = fb_ref.position[1]) THEN fb_ref.leave(); END_IF, VisuElemId=-1
    hotkey  Id=481037385728, Key=KeyDown=True, KeyName=down, ActionToExecute=Action=STSnippet=IF d_pad_pos[0] = fb_ref.position[0] AND d_pad_pos[1] = fb_ref.position[1] THEN fb_ref.select(); END_IF IF NOT(d_pad_pos[0] = fb_ref.position[0] AND d_pad_pos[1] = fb_ref.position[1]) THEN fb_ref.leave(); END_IF, VisuElemId=-1
    hotkey  Id=481041580032, Key=KeyName=SPACE, ActionToExecute=Action=STSnippet=IF d_pad_pos[0] = fb_ref.position[0] AND d_pad_pos[1] <> fb_ref.position[1] THEN fb_ref.close(); d_pad_pos[0]:= 0; d_pad_pos[1]:= 0; fb_ref.hover(); END_IF, VisuElemId=-1
END_VISUALIZATION

// ecomatDisplay43inch_64bit_1/Application/hmi/menu objects/menu data/Empty_visu_reference
VISUALIZATION Empty_visu_reference  // 1024x768
END_VISUALIZATION

// ecomatDisplay43inch_64bit_1/Application/hmi/menu objects/menu item/menu_item
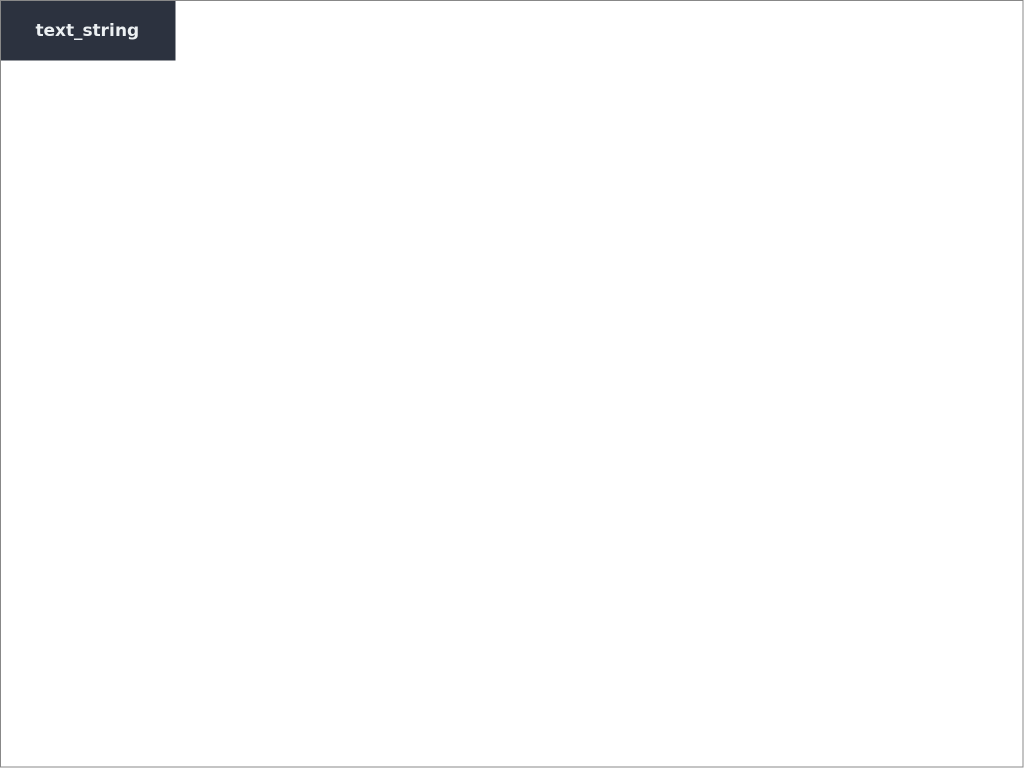
VISUALIZATION menu_item  // 1024x768
VAR_INPUT
	fb_ref: REFERENCE TO fb_menu_item;
	d_pad_pos: REFERENCE TO ARRAY [0..1] OF UINT;
END_VAR
    Image (118,3 52x52)
        p84334746: image_id
    Rectangle (0,0 175x60)
    Rectangle (0,0 175x60)
    Rectangle (0,0 175x60), colour variable: fb_ref.color
        p3450524324: fb_ref.color
        p3092690914: fb_ref.color
        p2167032090: fb_ref.color
        OnMouseClick: execute { fb_ref.select(); }
        OnMouseDown: execute {  }
        OnMouseEnter: execute { fb_ref.hover(); }
        OnMouseLeave: execute { fb_ref.leave(); }
    Rectangle (0,0 175x60), "text_string", text variable: text_string
    Rectangle (0,0 175x60), colour variable: fb_ref.color
        p3450524324: fb_ref.color
        p3092690914: fb_ref.color
        p2167032090: fb_ref.color
        OnMouseClick: execute {  }
        OnMouseDown: execute { fb_ref.select(); d_pad_pos:= fb_ref.position; }
        OnMouseEnter: execute { fb_ref.hover(); }
        OnMouseLeave: execute { fb_ref.leave(); }
        OnMouseUp: execute { fb_ref.hover(); }
    hotkey  Id=481037385728, Key=KeyName=SPACE, ActionToExecute=Action=STSnippet=IF d_pad_pos[0] = fb_ref.position[0] AND d_pad_pos[1] = fb_ref.position[1] THEN fb_ref.select(); fb_ref.item_action(); END_IF, VisuElemId=-1
    hotkey  Id=481038434304, Key=KeyDown=True, KeyName=right, ActionToExecute=Action=STSnippet=IF d_pad_pos[0] = fb_ref.position[0] AND d_pad_pos[1] = fb_ref.position[1] THEN fb_ref.hover(); END_IF IF NOT(d_pad_pos[0] = fb_ref.position[0] AND d_pad_pos[1] = fb_ref.position[1]) THEN fb_ref.leave(); END_IF, VisuElemId=-1
    hotkey  Id=481039482880, Key=KeyDown=True, KeyName=left, ActionToExecute=Action=STSnippet=IF d_pad_pos[0] = fb_ref.position[0] AND d_pad_pos[1] = fb_ref.position[1] THEN fb_ref.hover(); END_IF IF NOT(d_pad_pos[0] = fb_ref.position[0] AND d_pad_pos[1] = fb_ref.position[1]) THEN fb_ref.leave(); END_IF, VisuElemId=-1
    hotkey  Id=481040531456, Key=KeyDown=True, KeyName=up, ActionToExecute=Action=STSnippet=IF d_pad_pos[0] = fb_ref.position[0] AND d_pad_pos[1] = fb_ref.position[1] THEN fb_ref.hover(); fb_ref.item_action(); END_IF IF NOT(d_pad_pos[0] = fb_ref.position[0] AND d_pad_pos[1] = fb_ref.position[1]) THEN fb_ref.leave(); END_IF, VisuElemId=-1
    hotkey  Id=481041580032, Key=KeyDown=True, KeyName=down, ActionToExecute=Action=STSnippet=IF d_pad_pos[0] = fb_ref.position[0] AND d_pad_pos[1] = fb_ref.position[1] THEN fb_ref.hover(); fb_ref.item_action(); END_IF IF NOT(d_pad_pos[0] = fb_ref.position[0] AND d_pad_pos[1] = fb_ref.position[1]) THEN fb_ref.leave(); END_IF, VisuElemId=-1
END_VISUALIZATION

// ecomatDisplay43inch_64bit_1/Application/hmi/menu objects/toggle items/toggle_item
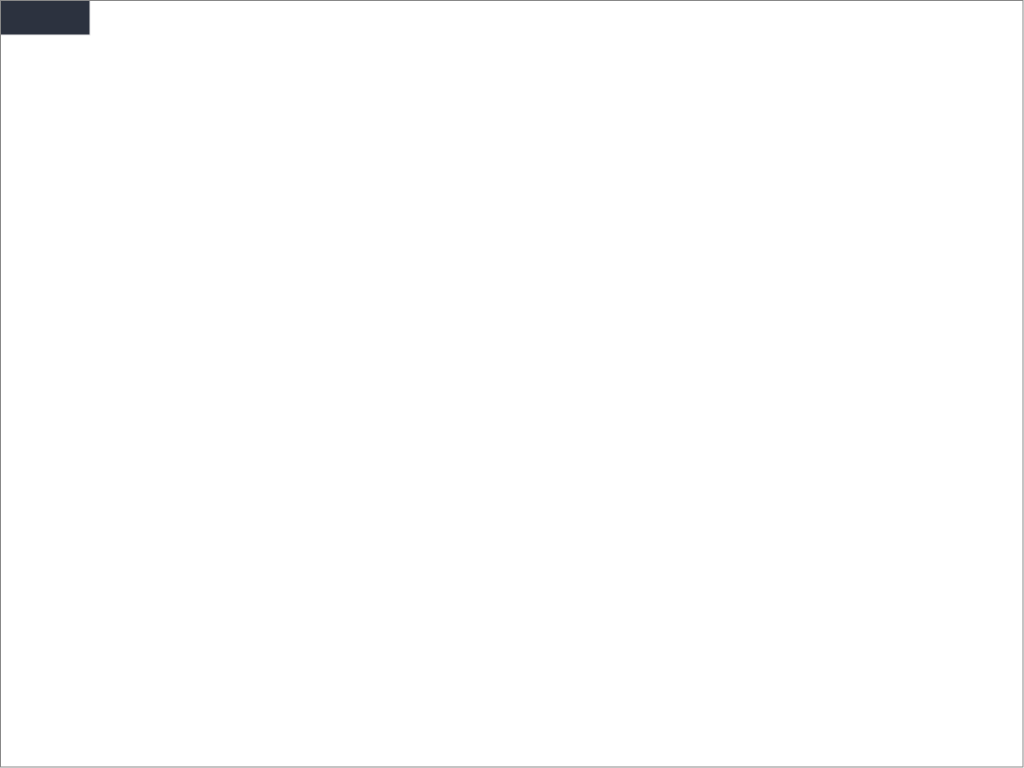
VISUALIZATION toggle_item  // 1024x768
VAR_INPUT
	fb_ref: REFERENCE TO fb_dummy_item;
	d_pad_pos: REFERENCE TO ARRAY [0..1] OF UINT;
END_VAR

VAR
	selected: BOOL;
END_VAR
    Rectangle (0,0 90x35)
    Rectangle (0,0 90x35)
    Rectangle (0,0 90x35), colour variable: fb_ref.color
        p3450524324: fb_ref.color
        p3092690914: fb_ref.color
        p2167032090: fb_ref.color
        OnMouseClick: execute { fb_ref.select(); }
        OnMouseDown: execute {  }
        OnMouseEnter: execute { fb_ref.hover(); }
        OnMouseLeave: execute { fb_ref.leave(); }
    Rectangle (0,0 90x35), colour toggle: fb_ref.color = g_menu_colors.nav[nav_item_enum.selected], colour variable: fb_ref.color
        p3450524324: g_menu_colors.nav[nav_item_enum.selected]
        p3092690914: g_menu_colors.nav[nav_item_enum.accent]
        p2167032090: fb_ref.color
        OnMouseClick: execute {  }
        OnMouseDown: execute {
            fb_ref.select();
            d_pad_pos:= fb_ref.position;
            selected:= 1;
        }
        OnMouseEnter: execute { fb_ref.hover(); }
        OnMouseLeave: execute { fb_ref.leave(); selected:= 0; }
        OnMouseUp: execute {  }
    hotkey  Id=481040531456, Key=KeyName=right, ActionToExecute=Action=STSnippet=IF d_pad_pos[0] = fb_ref.position[0] AND d_pad_pos[1] = fb_ref.position[1] THEN fb_ref.hover(); selected:= 1; END_IF IF NOT(d_pad_pos[0] = fb_ref.position[0] AND d_pad_pos[1] = fb_ref.position[1]) THEN fb_ref.leave(); selected:= 0; END_IF, VisuElemId=-1
    hotkey  Id=481039482880, Key=KeyName=left, ActionToExecute=Action=STSnippet=IF d_pad_pos[0] = fb_ref.position[0] AND d_pad_pos[1] = fb_ref.position[1] THEN fb_ref.hover(); selected:= 1; END_IF IF NOT(d_pad_pos[0] = fb_ref.position[0] AND d_pad_pos[1] = fb_ref.position[1]) THEN fb_ref.leave(); selected:= 0; END_IF, VisuElemId=-1
    hotkey  Id=481038434304, Key=KeyName=up, ActionToExecute=Action=STSnippet=IF d_pad_pos[0] = fb_ref.position[0] AND d_pad_pos[1] = fb_ref.position[1] THEN fb_ref.hover(); selected:= 1; END_IF IF NOT(d_pad_pos[0] = fb_ref.position[0] AND d_pad_pos[1] = fb_ref.position[1]) THEN fb_ref.leave(); selected:= 0; END_IF, VisuElemId=-1
    hotkey  Id=481037385728, Key=KeyName=down, ActionToExecute=Action=STSnippet=IF d_pad_pos[0] = fb_ref.position[0] AND d_pad_pos[1] = fb_ref.position[1] THEN fb_ref.hover(); selected:= 1; END_IF IF NOT(d_pad_pos[0] = fb_ref.position[0] AND d_pad_pos[1] = fb_ref.position[1]) THEN fb_ref.leave(); selected:= 0; END_IF, VisuElemId=-1
END_VISUALIZATION

// ecomatDisplay43inch_64bit_1/Application/hmi/menu objects/toggle items/integer setting/integer_setting_dialog
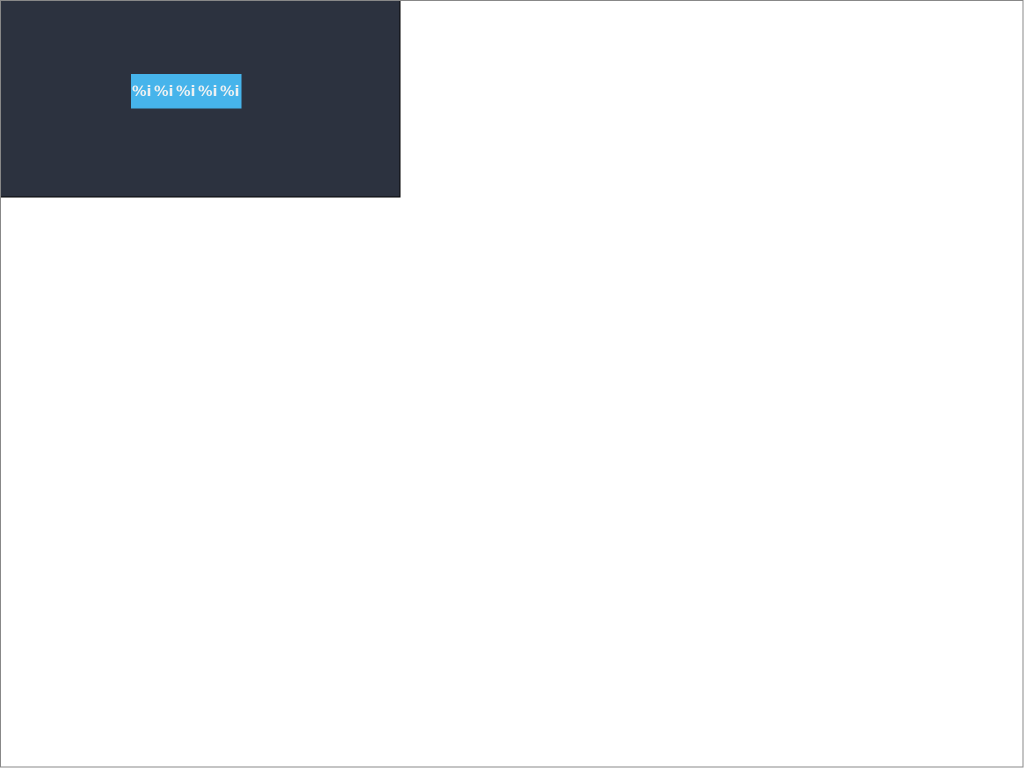
VISUALIZATION integer_setting_dialog  // 1024x768
VAR_INPUT
	fb_ref: REFERENCE TO fb_integer_setting;
	ref_d_pad: REFERENCE TO d_pad_fb;
END_VAR

VAR
	sel_d_pad: d_pad_fb:= (x_bounds:= 7);
END_VAR
    Rectangle (-4,-11 404x208), colour variable: g_menu_colors.default
        p3450524324: g_menu_colors.default
    Rectangle (131,74 22x34), "%i", text variable: (fb_ref.integer / 10000) MOD 10, colour toggle: sel_d_pad.position[0] = 5, colour variable: 16#FF2C323F
        p3450524324: 16#FF2C323F
        p3092690914: 16#FF46B4EB
        p2167032090: 16#FF46B4EB
        OnMouseClick: execute { fb_ref.select(); }
        OnMouseDown: execute {  }
        OnMouseEnter: execute { fb_ref.hover(); }
        OnMouseLeave: execute { fb_ref.leave(); }
    Rectangle (153,74 22x34), "%i", text variable: (fb_ref.integer / 1000) MOD 10, colour toggle: sel_d_pad.position[0] = 4, colour variable: 16#FF2C323F
        p3450524324: 16#FF2C323F
        p3092690914: 16#FF46B4EB
        p2167032090: 16#FF46B4EB
        OnMouseClick: execute { fb_ref.select(); }
        OnMouseDown: execute {  }
        OnMouseEnter: execute { fb_ref.hover(); }
        OnMouseLeave: execute { fb_ref.leave(); }
    Rectangle (175,74 22x34), "%i", text variable: (fb_ref.integer / 100) MOD 10, colour toggle: sel_d_pad.position[0] = 3, colour variable: 16#FF2C323F
        p3450524324: 16#FF2C323F
        p3092690914: 16#FF46B4EB
        p2167032090: 16#FF46B4EB
        OnMouseClick: execute { fb_ref.select(); }
        OnMouseDown: execute {  }
        OnMouseEnter: execute { fb_ref.hover(); }
        OnMouseLeave: execute { fb_ref.leave(); }
    Rectangle (197,74 22x34), "%i", text variable: (fb_ref.integer / 10) MOD 10, colour toggle: sel_d_pad.position[0] = 2, colour variable: 16#FF2C323F
        p3450524324: 16#FF2C323F
        p3092690914: 16#FF46B4EB
        p2167032090: 16#FF46B4EB
        OnMouseClick: execute { fb_ref.select(); }
        OnMouseDown: execute {  }
        OnMouseEnter: execute { fb_ref.hover(); }
        OnMouseLeave: execute { fb_ref.leave(); }
    Rectangle (219,74 22x34), "%i", text variable: (fb_ref.integer) MOD 10, colour toggle: sel_d_pad.position[0] = 1, colour variable: 16#FF2C323F
        p3450524324: 16#FF2C323F
        p3092690914: 16#FF46B4EB
        p2167032090: 16#FF46B4EB
        OnMouseClick: execute { fb_ref.select(); }
        OnMouseDown: execute {  }
        OnMouseEnter: execute { fb_ref.hover(); }
        OnMouseLeave: execute { fb_ref.leave(); }
    hotkey  Id=481041580032, Key=KeyName=right, ActionToExecute=Action=STSnippet=IF fb_ref.selected THEN sel_d_pad.right(); RETURN; END_IF IF ref_d_pad.position[0] = fb_ref.position[0] AND ref_d_pad.position[1] = fb_ref.position[1] THEN fb_ref.hover(); END_IF IF NOT(ref_d_pad.position[0] = fb_ref.position[0] AND ref_d_pad.position[1] = fb_ref.position[1]) THEN fb_ref.leave(); END_IF, VisuElemId=-1
    hotkey  Id=481040531456, Key=KeyName=left, ActionToExecute=Action=STSnippet=IF fb_ref.selected THEN sel_d_pad.left(); RETURN; END_IF IF ref_d_pad.position[0] = fb_ref.position[0] AND ref_d_pad.position[1] = fb_ref.position[1] THEN fb_ref.hover(); END_IF IF NOT(ref_d_pad.position[0] = fb_ref.position[0] AND ref_d_pad.position[1] = fb_ref.position[1]) THEN fb_ref.leave(); END_IF, VisuElemId=-1
    hotkey  Id=481039482880, Key=KeyName=up, ActionToExecute=Action=STSnippet=IF fb_ref.selected THEN fb_ref.increase(); RETURN; END_IF IF ref_d_pad.position[0] = fb_ref.position[0] AND ref_d_pad.position[1] = fb_ref.position[1] THEN fb_ref.hover(); END_IF IF NOT(ref_d_pad.position[0] = fb_ref.position[0] AND ref_d_pad.position[1] = fb_ref.position[1]) THEN fb_ref.leave(); END_IF, VisuElemId=-1
    hotkey  Id=481038434304, Key=KeyName=down, ActionToExecute=Action=STSnippet=IF fb_ref.selected THEN fb_ref.decrease(); RETURN; END_IF IF ref_d_pad.position[0] = fb_ref.position[0] AND ref_d_pad.position[1] = fb_ref.position[1] THEN fb_ref.hover(); END_IF IF NOT(ref_d_pad.position[0] = fb_ref.position[0] AND ref_d_pad.position[1] = fb_ref.position[1]) THEN fb_ref.leave(); END_IF, VisuElemId=-1
    hotkey  Id=481037385728, Key=KeyName=space, ActionToExecute=Action=STSnippet=IF fb_ref.position[0] = ref_d_pad.position[0] AND fb_ref.position[1] = ref_d_pad.position[1] THEN fb_ref.select(); ref_d_pad.disable_nav:= ref_d_pad.disable_nav XOR TRUE; END_IF, VisuElemId=-1
END_VISUALIZATION

// ecomatDisplay43inch_64bit_1/Application/hmi/menu objects/toggle items/integer setting/integer_setting_item
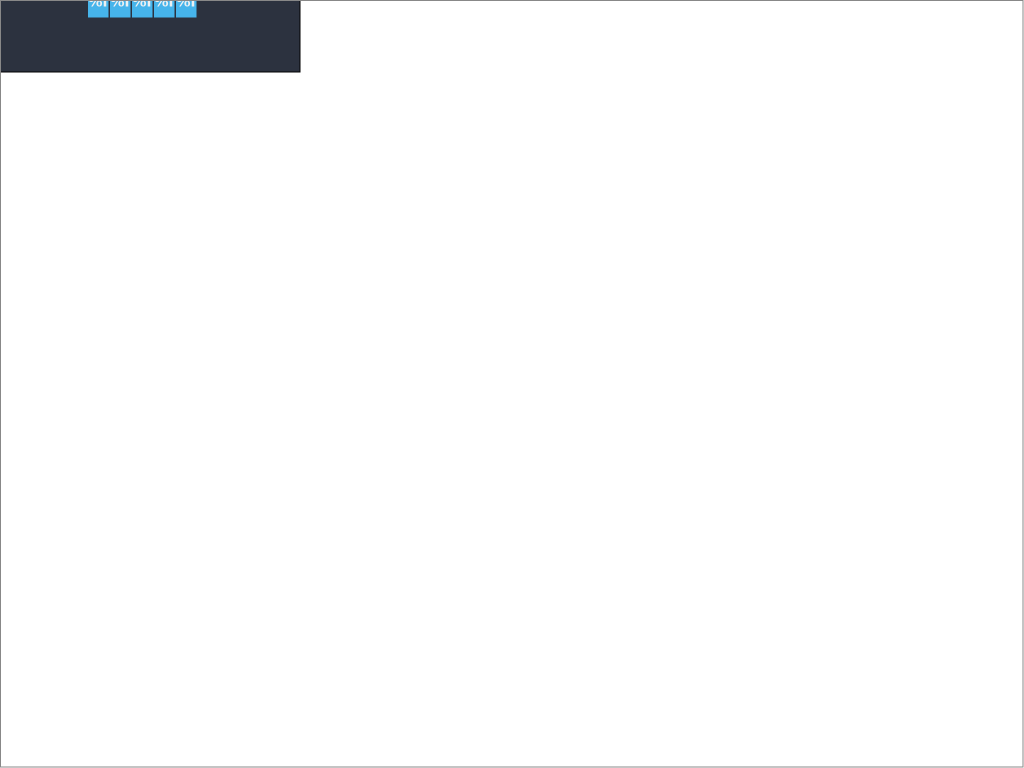
VISUALIZATION integer_setting_item  // 1024x768
VAR_INPUT
	fb_ref: REFERENCE TO fb_integer_setting;
	ref_d_pad: REFERENCE TO d_pad_fb;
END_VAR

VAR
	sel_d_pad: d_pad_fb:= (x_bounds:= 7);
END_VAR
    Rectangle (0,0 300x45), invisible if: ref_d_pad.disable_nav
    Rectangle (0,0 300x45), invisible if: ref_d_pad.disable_nav
    Rectangle (0,0 300x45), invisible if: ref_d_pad.disable_nav, colour variable: fb_ref.color
        p3450524324: fb_ref.color
        p3092690914: fb_ref.color
        p2167032090: fb_ref.color
        OnMouseClick: execute { fb_ref.select(); }
        OnMouseDown: execute {  }
        OnMouseEnter: execute { fb_ref.hover(); }
        OnMouseLeave: execute { fb_ref.leave(); }
    Rectangle (0,0 300x45), colour toggle: fb_ref.color = g_menu_colors.nav[nav_item_enum.selected], invisible if: ref_d_pad.disable_nav, colour variable: fb_ref.color
        p3450524324: g_menu_colors.nav[nav_item_enum.selected]
        p3092690914: g_menu_colors.nav[nav_item_enum.accent]
        p2167032090: fb_ref.color
        OnMouseClick: execute {  }
        OnMouseDown: execute { fb_ref.select(); ref_d_pad.position:= fb_ref.position; }
        OnMouseEnter: execute { fb_ref.hover(); }
        OnMouseLeave: execute { fb_ref.leave(); ref_d_pad.disable_nav:= 0; }
        OnMouseUp: execute {  }
    Rectangle (14,5 160x34), "%s", text variable: st_name, invisible if: ref_d_pad.disable_nav
        OnMouseClick: execute { fb_ref.select(); }
        OnMouseDown: execute {  }
        OnMouseEnter: execute { fb_ref.hover(); }
        OnMouseLeave: execute { fb_ref.leave(); }
    Rectangle (170,5 60x34), "%i", text variable: fb_ref.integer, invisible if: ref_d_pad.disable_nav
        OnMouseClick: execute { fb_ref.select(); }
        OnMouseDown: execute {  }
        OnMouseEnter: execute { fb_ref.hover(); }
        OnMouseLeave: execute { fb_ref.leave(); }
    Rectangle (237,5 53x34), "%s", text variable: st_units, invisible if: ref_d_pad.disable_nav
        OnMouseClick: execute { fb_ref.select(); }
        OnMouseDown: execute {  }
        OnMouseEnter: execute { fb_ref.hover(); }
        OnMouseLeave: execute { fb_ref.leave(); }
    Rectangle (0,-72 300x144), invisible if: NOT(fb_ref.selected), colour variable: g_menu_colors.default
        p3450524324: g_menu_colors.default
    Rectangle (87,-16 22x34), "%i", text variable: (fb_ref.integer / 10000) MOD 10, colour toggle: sel_d_pad.position[0] = 5, invisible if: NOT(fb_ref.selected), colour variable: 16#FF2C323F
        p3450524324: 16#FF2C323F
        p3092690914: 16#FF46B4EB
        p2167032090: 16#FF46B4EB
        OnMouseClick: execute { fb_ref.select(); }
        OnMouseDown: execute {  }
        OnMouseEnter: execute { fb_ref.hover(); }
        OnMouseLeave: execute { fb_ref.leave(); }
    Rectangle (109,-16 22x34), "%i", text variable: (fb_ref.integer / 1000) MOD 10, colour toggle: sel_d_pad.position[0] = 4, invisible if: NOT(fb_ref.selected), colour variable: 16#FF2C323F
        p3450524324: 16#FF2C323F
        p3092690914: 16#FF46B4EB
        p2167032090: 16#FF46B4EB
        OnMouseClick: execute { fb_ref.select(); }
        OnMouseDown: execute {  }
        OnMouseEnter: execute { fb_ref.hover(); }
        OnMouseLeave: execute { fb_ref.leave(); }
    Rectangle (131,-16 22x34), "%i", text variable: (fb_ref.integer / 100) MOD 10, colour toggle: sel_d_pad.position[0] = 3, invisible if: NOT(fb_ref.selected), colour variable: 16#FF2C323F
        p3450524324: 16#FF2C323F
        p3092690914: 16#FF46B4EB
        p2167032090: 16#FF46B4EB
        OnMouseClick: execute { fb_ref.select(); }
        OnMouseDown: execute {  }
        OnMouseEnter: execute { fb_ref.hover(); }
        OnMouseLeave: execute { fb_ref.leave(); }
    Rectangle (153,-16 22x34), "%i", text variable: (fb_ref.integer / 10) MOD 10, colour toggle: sel_d_pad.position[0] = 2, invisible if: NOT(fb_ref.selected), colour variable: 16#FF2C323F
        p3450524324: 16#FF2C323F
        p3092690914: 16#FF46B4EB
        p2167032090: 16#FF46B4EB
        OnMouseClick: execute { fb_ref.select(); }
        OnMouseDown: execute {  }
        OnMouseEnter: execute { fb_ref.hover(); }
        OnMouseLeave: execute { fb_ref.leave(); }
    Rectangle (175,-16 22x34), "%i", text variable: (fb_ref.integer) MOD 10, colour toggle: sel_d_pad.position[0] = 1, invisible if: NOT(fb_ref.selected), colour variable: 16#FF2C323F
        p3450524324: 16#FF2C323F
        p3092690914: 16#FF46B4EB
        p2167032090: 16#FF46B4EB
        OnMouseClick: execute { fb_ref.select(); }
        OnMouseDown: execute {  }
        OnMouseEnter: execute { fb_ref.hover(); }
        OnMouseLeave: execute { fb_ref.leave(); }
    hotkey  Id=481040531456, Key=KeyName=right, ActionToExecute=Action=STSnippet=IF fb_ref.selected THEN sel_d_pad.right(); RETURN; END_IF IF ref_d_pad.position[0] = fb_ref.position[0] AND ref_d_pad.position[1] = fb_ref.position[1] THEN fb_ref.hover(); END_IF IF NOT(ref_d_pad.position[0] = fb_ref.position[0] AND ref_d_pad.position[1] = fb_ref.position[1]) THEN fb_ref.leave(); END_IF, VisuElemId=-1
    hotkey  Id=481039482880, Key=KeyName=left, ActionToExecute=Action=STSnippet=IF fb_ref.selected THEN sel_d_pad.left(); RETURN; END_IF IF ref_d_pad.position[0] = fb_ref.position[0] AND ref_d_pad.position[1] = fb_ref.position[1] THEN fb_ref.hover(); END_IF IF NOT(ref_d_pad.position[0] = fb_ref.position[0] AND ref_d_pad.position[1] = fb_ref.position[1]) THEN fb_ref.leave(); END_IF, VisuElemId=-1
    hotkey  Id=481038434304, Key=KeyName=up, ActionToExecute=Action=STSnippet=IF fb_ref.selected AND fb_ref.integer + TO_UINT(EXPT(10, sel_d_pad.position[0] - 1)) <= fb_ref.max_value THEN fb_ref.integer:= fb_ref.integer + TO_UINT(EXPT(10, sel_d_pad.position[0] - 1)); RETURN; END_IF IF ref_d_pad.position[0] = fb_ref.position[0] AND ref_d_pad.position[1] = fb_ref.position[1] THEN fb_ref.hover(); END_IF IF NOT(ref_d_pad.position[0] = fb_ref.position[0] AND ref_d_pad.position[1] = fb_ref.position[1]) THEN fb_ref.leave(); END_IF, VisuElemId=-1
    hotkey  Id=481037385728, Key=KeyName=down, ActionToExecute=Action=STSnippet=IF fb_ref.selected AND fb_ref.integer - TO_UINT(EXPT(10, sel_d_pad.position[0] - 1)) >= fb_ref.min_value AND fb_ref.integer - TO_UINT(EXPT(10, sel_d_pad.position[0] - 1)) <= fb_ref.max_value THEN fb_ref.integer:= fb_ref.integer - TO_UINT(EXPT(10, sel_d_pad.position[0] - 1)); RETURN; END_IF IF ref_d_pad.position[0] = fb_ref.position[0] AND ref_d_pad.position[1] = fb_ref.position[1] THEN fb_ref.hover(); END_IF IF NOT(ref_d_pad.position[0] = fb_ref.position[0] AND ref_d_pad.position[1] = fb_ref.position[1]) THEN fb_ref.leave(); END_IF, VisuElemId=-1
    hotkey  Id=481041580032, Key=KeyName=space, ActionToExecute=Action=STSnippet=IF fb_ref.position[0] = ref_d_pad.position[0] AND fb_ref.position[1] = ref_d_pad.position[1] THEN fb_ref.select(); ref_d_pad.disable_nav:= ref_d_pad.disable_nav XOR TRUE; END_IF, VisuElemId=-1
END_VISUALIZATION

// ecomatDisplay43inch_64bit_1/Application/hmi/menu objects/toggle items/real setting/real_setting_item
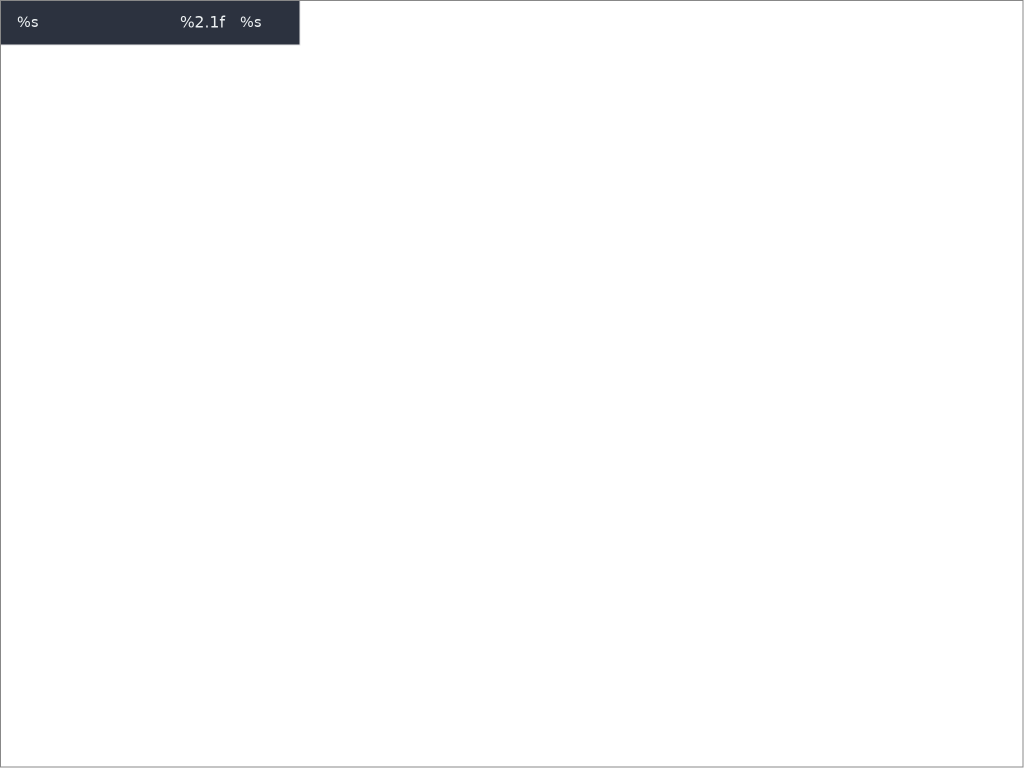
VISUALIZATION real_setting_item  // 1024x768
VAR_INPUT
	fb_ref: REFERENCE TO fb_real_setting;
	ref_d_pad: REFERENCE TO d_pad_fb;
END_VAR
    Rectangle (0,0 300x45)
    Rectangle (0,0 300x45)
    Rectangle (0,0 300x45), colour variable: fb_ref.color
        p3450524324: fb_ref.color
        p3092690914: fb_ref.color
        p2167032090: fb_ref.color
        OnMouseClick: execute { fb_ref.select(); }
        OnMouseDown: execute {  }
        OnMouseEnter: execute { fb_ref.hover(); }
        OnMouseLeave: execute { fb_ref.leave(); }
    Rectangle (0,0 300x45), colour toggle: fb_ref.color = g_menu_colors.nav[nav_item_enum.selected], colour variable: fb_ref.color
        p3450524324: g_menu_colors.nav[nav_item_enum.selected]
        p3092690914: g_menu_colors.nav[nav_item_enum.accent]
        p2167032090: fb_ref.color
        OnMouseClick: execute {  }
        OnMouseDown: execute { fb_ref.select(); ref_d_pad.position:= fb_ref.position; }
        OnMouseEnter: execute { fb_ref.hover(); }
        OnMouseLeave: execute { fb_ref.leave(); ref_d_pad.disable_nav:= 0; }
        OnMouseUp: execute {  }
    Rectangle (14,5 160x34), "%s", text variable: st_name
        OnMouseClick: execute { fb_ref.select(); }
        OnMouseDown: execute {  }
        OnMouseEnter: execute { fb_ref.hover(); }
        OnMouseLeave: execute { fb_ref.leave(); }
    Rectangle (170,5 58x34), "%2.1f", text variable: fb_ref.real_var
        OnMouseClick: execute { fb_ref.select(); }
        OnMouseDown: execute {  }
        OnMouseEnter: execute { fb_ref.hover(); }
        OnMouseLeave: execute { fb_ref.leave(); }
    Rectangle (237,5 43x34), "%s", text variable: st_units
        OnMouseClick: execute { fb_ref.select(); }
        OnMouseDown: execute {  }
        OnMouseEnter: execute { fb_ref.hover(); }
        OnMouseLeave: execute { fb_ref.leave(); }
    hotkey  Id=481040531456, Key=KeyName=right, ActionToExecute=Action=STSnippet=IF fb_ref.selected THEN RETURN; END_IF IF ref_d_pad.position[0] = fb_ref.position[0] AND ref_d_pad.position[1] = fb_ref.position[1] THEN fb_ref.hover(); END_IF IF NOT(ref_d_pad.position[0] = fb_ref.position[0] AND ref_d_pad.position[1] = fb_ref.position[1]) THEN fb_ref.leave(); END_IF, VisuElemId=-1
    hotkey  Id=481039482880, Key=KeyName=left, ActionToExecute=Action=STSnippet=IF fb_ref.selected THEN RETURN; END_IF IF ref_d_pad.position[0] = fb_ref.position[0] AND ref_d_pad.position[1] = fb_ref.position[1] THEN fb_ref.hover(); END_IF IF NOT(ref_d_pad.position[0] = fb_ref.position[0] AND ref_d_pad.position[1] = fb_ref.position[1]) THEN fb_ref.leave(); END_IF, VisuElemId=-1
    hotkey  Id=481038434304, Key=KeyName=up, ActionToExecute=Action=STSnippet=IF fb_ref.selected THEN fb_ref.increase(); RETURN; END_IF IF ref_d_pad.position[0] = fb_ref.position[0] AND ref_d_pad.position[1] = fb_ref.position[1] THEN fb_ref.hover(); END_IF IF NOT(ref_d_pad.position[0] = fb_ref.position[0] AND ref_d_pad.position[1] = fb_ref.position[1]) THEN fb_ref.leave(); END_IF, VisuElemId=-1
    hotkey  Id=481037385728, Key=KeyName=down, ActionToExecute=Action=STSnippet=IF fb_ref.selected THEN fb_ref.decrease(); RETURN; END_IF IF ref_d_pad.position[0] = fb_ref.position[0] AND ref_d_pad.position[1] = fb_ref.position[1] THEN fb_ref.hover(); END_IF IF NOT(ref_d_pad.position[0] = fb_ref.position[0] AND ref_d_pad.position[1] = fb_ref.position[1]) THEN fb_ref.leave(); END_IF, VisuElemId=-1
    hotkey  Id=481041580032, Key=KeyName=space, ActionToExecute=Action=STSnippet=IF fb_ref.position[0] = ref_d_pad.position[0] AND fb_ref.position[1] = ref_d_pad.position[1] THEN fb_ref.select(); ref_d_pad.disable_nav:= ref_d_pad.disable_nav XOR TRUE; END_IF, VisuElemId=-1
END_VISUALIZATION
